// TIA Portal V20 export
DATA_BLOCK "DB_ConveyorParameters"   // DB26
// stored: Access Published, MemoryReserve 100, Namespace LineB1
   VAR
      Line : Struct
         B1 : Struct
            Conveyor : Array[_.minB1.._.maxB1] of "LineB1.ConveyorParameters";
         END_STRUCT;
      END_STRUCT;
   END_VAR
BEGIN
END_DATA_BLOCK
